Yaskawa INFORM job: X2_24B(90,0).JBI

/JOB
//NAME X2_24B(90,0)
///FOLDERNAME X2
//POS
///NPOS 98,98,98,6,0,0
///TOOL 0
///POSTYPE PULSE
///PULSE
C00000=15575,79859,-14986,13441,104676,73483
C00001=126804,-92055,-48789,28645,51065,65926
C00002=154512,-17095,-20441,46457,51312,77671
C00003=161937,-848,-6352,37251,32753,61979
C00004=159692,17407,12655,41702,31966,59656
C00005=159970,19766,16047,42399,31172,59288
C00006=159972,20330,18267,43630,30372,58648
C00007=159976,20326,18034,43461,30475,58736
C00008=160482,23050,20629,43221,30080,58863
C00009=159976,20326,18034,43461,30475,58736
C00010=159697,17919,14587,42706,31268,59129
C00011=158976,12160,6349,41128,33206,59971
C00012=159418,6486,-154,59703,53174,49617
C00013=160929,10789,6591,60497,51224,48988
C00014=161518,12599,9400,60873,50446,48712
C00015=161521,13127,11564,61641,49913,48166
C00016=161520,13051,11326,61563,49966,48222
C00017=162429,14896,13007,61347,49349,48376
C00018=161520,13051,11326,61563,49966,48222
C00019=160931,11199,8471,61161,50742,48508
C00020=159420,6798,1623,60306,52686,49160
C00021=158595,11215,4105,55963,68819,69684
C00022=160652,12318,8052,56162,66520,69358
C00023=161472,12850,9720,56269,65597,69221
C00024=161473,13383,11888,56662,64989,68781
C00025=161490,13285,11447,56576,65106,68876
C00026=162644,13596,11726,56360,64407,69116
C00027=161490,13285,11447,56576,65106,68876
C00028=160670,12719,9745,56453,66030,69019
C00029=158615,11533,5714,56217,68333,69354
C00030=145844,21981,14022,59749,100145,59975
C00031=147472,19762,14879,59544,98258,59599
C00032=148136,18948,15302,59481,97487,59448
C00033=148138,19507,17514,59327,96919,59020
C00034=148144,19438,17214,59348,96993,59081
C00035=149095,17801,15678,59427,96459,59294
C00036=148144,19438,17214,59348,96993,59081
C00037=147479,20220,16761,59400,97767,59232
C00038=145852,22359,15824,59578,99660,59607
C00039=137889,24717,18086,55155,118108,53390
C00040=138207,19130,15660,54565,117103,52873
C00041=138207,19573,17388,54175,116602,52518
C00042=138207,19438,16874,54289,116751,52623
C00043=138402,17218,14803,54401,116718,52725
C00044=138207,19198,15931,54502,117024,52816
C00045=138380,23714,17318,55251,117790,53487
C00046=145852,22359,15824,59578,99660,59607
C00047=154763,11901,15387,68658,70711,41061
C00048=156717,15177,21386,69242,68625,40420
C00049=157143,15546,21805,69251,68310,40447
C00050=156255,14972,22417,69511,68656,40020
C00051=157248,16273,23616,69515,67962,40120
C00052=157236,16335,23673,69517,67969,40117
C00053=158136,15421,22899,68081,54770,43017
C00054=158597,17339,24094,63812,43421,46704
C00055=158675,18696,25754,61305,36586,48793
C00056=158371,15338,21521,60414,37218,49285
C00057=157215,9529,13249,58606,39045,50279
C00058=155689,128,-5597,51101,67034,60953
C00059=149151,12252,4951,55421,100768,64918
C00060=144904,3935,5079,54220,100687,62374
C00061=145543,-5451,3457,53674,97956,61056
C00062=145117,-2050,7462,53507,97767,60700
C00063=146427,-4037,5767,53710,97024,60980
C00064=153396,2613,11325,54625,92971,62406
C00065=155096,3131,11794,54961,91043,63070
C00066=155127,3166,11823,54964,91024,63076
C00067=158177,1489,10598,55836,83437,65573
C00068=162825,5929,14207,55721,72913,69138
C00069=166488,10840,18435,54134,62935,72728
C00070=165195,8380,15225,53946,63632,72915
C00071=163039,7025,11023,53573,66027,73191
C00072=156115,13997,17270,60701,43178,45173
C00073=157268,19891,25768,62434,41355,44161
C00074=157884,21006,27154,62518,40826,44139
C00075=156967,20197,27277,63317,41176,43618
C00076=158134,20809,27857,62990,40410,43871
C00077=158121,20875,27920,62999,40416,43865
C00078=157099,23447,30366,63399,40803,43589
C00079=155705,26353,33233,56778,30914,48004
C00080=155359,26555,33368,49384,25433,52187
C00081=153014,28261,34997,43179,22329,55472
C00082=153895,25102,30778,39953,22434,57086
C00083=153561,18171,21135,36977,24464,58522
C00084=154328,-437,-7083,34814,53153,69175
C00085=153943,-3670,1993,58187,73110,66585
C00086=156220,-2957,5589,58514,70714,66272
C00087=156644,-2599,7283,58737,69991,66002
C00088=157747,-4828,5565,58281,66085,67202
C00089=157731,-4759,5622,58282,66096,67199
C00090=159511,-232,9113,57226,61670,68810
C00091=163403,5947,13806,51963,49845,73894
C00092=165030,15735,22851,46781,40971,78339
C00093=162686,15609,21777,49814,45504,76092
C00094=160796,11946,15422,49130,47880,76469
C00095=139502,-13197,-17498,52190,59618,73701
C00096=102643,-76138,-42592,31929,63319,59034
C00097=-2000,-92055,-48789,0,51065,0
BC00000=67030,600285,936124
BC00001=198867,566215,454485
BC00002=198867,436418,248072
BC00003=170083,400556,144661
BC00004=170083,415917,144661
BC00005=170083,415917,144661
BC00006=170083,415917,144661
BC00007=170083,415917,144661
BC00008=170083,415917,144661
BC00009=170083,415917,144661
BC00010=170083,415917,144661
BC00011=170083,415917,144661
BC00012=170307,416366,144512
BC00013=170307,416366,144512
BC00014=170307,416366,144512
BC00015=170307,416366,144512
BC00016=170307,416366,144512
BC00017=170307,416366,144512
BC00018=170307,416366,144512
BC00019=170307,416366,144512
BC00020=170307,416366,144512
BC00021=173994,440513,186920
BC00022=173994,440513,186920
BC00023=173994,440513,186920
BC00024=173994,440513,186920
BC00025=173994,440513,186920
BC00026=173994,440513,186920
BC00027=173994,440513,186920
BC00028=173994,440513,186920
BC00029=173994,440513,186920
BC00030=162509,461304,186551
BC00031=162509,461304,186551
BC00032=162509,461304,186551
BC00033=162509,461304,186551
BC00034=162509,461304,186551
BC00035=162509,461304,186551
BC00036=162509,461304,186551
BC00037=162509,461304,186551
BC00038=162509,461304,186551
BC00039=162509,461304,186551
BC00040=162509,461304,186551
BC00041=162509,461304,186551
BC00042=162509,461304,186551
BC00043=162509,461304,186551
BC00044=162509,461304,186551
BC00045=162509,461304,186551
BC00046=162509,461304,186551
BC00047=159532,415917,202070
BC00048=159532,415917,202070
BC00049=159532,415917,202070
BC00050=159532,415917,202070
BC00051=159532,415917,202070
BC00052=159532,415917,202070
BC00053=159532,415917,202070
BC00054=159533,415917,202067
BC00055=159533,415917,202065
BC00056=159532,415917,202070
BC00057=159532,415917,202070
BC00058=177632,434837,235106
BC00059=187185,446552,262931
BC00060=187185,446552,262931
BC00061=187185,446551,262928
BC00062=187185,446551,262928
BC00063=187185,446551,262928
BC00064=187185,446551,262928
BC00065=187185,446552,262930
BC00066=187185,446552,262930
BC00067=187185,446552,262931
BC00068=187185,446552,262931
BC00069=187185,446552,262931
BC00070=187185,446552,262931
BC00071=187185,446552,262931
BC00072=161256,415917,204708
BC00073=161256,415917,204708
BC00074=161256,415917,204708
BC00075=161256,415917,204708
BC00076=161256,415917,204708
BC00077=161256,415917,204708
BC00078=161256,415917,204708
BC00079=161256,415917,204708
BC00080=161256,415917,204708
BC00081=161256,415917,204708
BC00082=161256,415917,204708
BC00083=161256,415917,204708
BC00084=162450,435407,231402
BC00085=163438,443373,249285
BC00086=163438,443373,249285
BC00087=163438,443373,249285
BC00088=163438,443373,249285
BC00089=163438,443373,249285
BC00090=163437,443372,249283
BC00091=163437,443372,249282
BC00092=163437,443372,249282
BC00093=163438,443373,249285
BC00094=163438,443373,249285
BC00095=167011,451779,248072
BC00096=167011,535447,454485
BC00097=198867,523905,632202
EC00000=-798151,-183836
EC00001=-798156,-183832
EC00002=-798156,-183832
EC00003=-798156,-183832
EC00004=-798156,-183832
EC00005=-798156,-183832
EC00006=-798156,-183832
EC00007=-798156,-183832
EC00008=-798156,-183832
EC00009=-798156,-183832
EC00010=-798156,-183832
EC00011=-798156,-183832
EC00012=-798156,-183832
EC00013=-798156,-183832
EC00014=-798156,-183832
EC00015=-798156,-183832
EC00016=-798156,-183832
EC00017=-798156,-183832
EC00018=-798156,-183832
EC00019=-798156,-183832
EC00020=-798156,-183832
EC00021=-798156,-183832
EC00022=-798156,-183832
EC00023=-798156,-183832
EC00024=-798156,-183832
EC00025=-798156,-183832
EC00026=-798156,-183832
EC00027=-798156,-183832
EC00028=-798156,-183832
EC00029=-798156,-183832
EC00030=-798156,-183832
EC00031=-798156,-183832
EC00032=-798156,-183832
EC00033=-798156,-183832
EC00034=-798156,-183832
EC00035=-798156,-183832
EC00036=-798156,-183832
EC00037=-798156,-183832
EC00038=-798156,-183832
EC00039=-798156,-183832
EC00040=-798156,-183832
EC00041=-798156,-183832
EC00042=-798156,-183832
EC00043=-798156,-183832
EC00044=-798156,-183832
EC00045=-798156,-183832
EC00046=-798156,-183832
EC00047=-798156,-183832
EC00048=-798156,-183832
EC00049=-798156,-183832
EC00050=-798156,-183832
EC00051=-798156,-183832
EC00052=-798156,-183832
EC00053=-798156,-183832
EC00054=-798155,-183833
EC00055=-798154,-183833
EC00056=-798156,-183832
EC00057=-798156,-183832
EC00058=-798156,-183832
EC00059=-798156,-183832
EC00060=-798156,-183832
EC00061=-798154,-183833
EC00062=-798154,-183833
EC00063=-798154,-183833
EC00064=-798154,-183833
EC00065=-798155,-183832
EC00066=-798155,-183832
EC00067=-798156,-183832
EC00068=-798156,-183832
EC00069=-798156,-183832
EC00070=-798156,-183832
EC00071=-798156,-183832
EC00072=-798156,-183832
EC00073=-798156,-183832
EC00074=-798156,-183832
EC00075=-798156,-183832
EC00076=-798156,-183832
EC00077=-798156,-183832
EC00078=-798156,-183832
EC00079=-798156,-183832
EC00080=-798156,-183832
EC00081=-798156,-183832
EC00082=-798156,-183832
EC00083=-798156,-183832
EC00084=-798156,-183832
EC00085=-798156,-183832
EC00086=-798156,-183832
EC00087=-798156,-183832
EC00088=-798156,-183832
EC00089=-798156,-183832
EC00090=-798156,-183832
EC00091=-798156,-183832
EC00092=-798156,-183832
EC00093=-798156,-183832
EC00094=-798156,-183832
EC00095=-798156,-183832
EC00096=-798156,-183832
EC00097=-798156,-183832
///POSTYPE BASE
///RECTAN
///RCONF 0,0,0,0,1,0,0,0,0,0,0,0,0,0,0,0,0,0,0,0,0,0,0,0
P00006=2.006,1.622,-0.565,0.0000,0.0000,0.0000
P00021=0.073,2.058,-0.109,0.0000,0.0000,0.0000
P00022=2.006,1.622,-0.565,0.0000,0.0000,0.0000
///RCONF 0,0,0,0,0,0,0,0,0,0,0,0,0,0,0,0,0,0,0,0,0,0,0,0
P00023=-2.957,-4.083,2.762,0.0000,0.0000,0.0000
P00024=-1.466,-0.226,-0.419,0.0000,0.0000,0.0000
P00030=-0.014,-0.768,0.131,0.0000,0.0000,0.0000
//INST
///DATE 2024/12/03 14:06
///ATTR SC,RW
///GROUP1 RB1,BS1
///GROUP2 ST1
NOP
'X2_24B(90,0)
MOVJ C00000 BC00000 VJ=100.00  +MOVJ EC00000 VJ=100.00
MOVJ C00001 BC00001 VJ=100.00  +MOVJ EC00001 VJ=100.00
MOVJ C00002 BC00002 VJ=100.00  +MOVJ EC00002 VJ=100.00
'Path S4187
SSFTOF
SFTOF3D
MOVJ C00003 BC00003 VJ=100.00  +MOVJ EC00003 VJ=100.00
MOVL C00004 BC00004 V=800.0  +MOVJ EC00004 VJ=100.00
SMOVL C00005 BC00005 V=166.7  +MOVJ EC00005
SREFP 3 C00006 BC00006  +REFP EC00006
CALL JOB:SEARCH-R1-S13D
SET P021 P006
SFTON3D P021
SMOVL C00007 BC00007 V=166.7  +MOVJ EC00007
SREFP 3 C00008 BC00008  +REFP EC00008
CALL JOB:SEARCH-R1-S13D
SET P021 P006
SMOVL C00009 BC00009 V=166.7  +MOVJ EC00009
MOVL C00010 BC00010 V=800.0  +MOVJ EC00010 VJ=100.00
MOVL C00011 BC00011 V=1000.0  +MOVJ EC00011 VJ=100.00
'EndPath S4187
'Path S4188
SFTOF3D
MOVJ C00012 BC00012 VJ=100.00  +MOVJ EC00012 VJ=100.00
MOVL C00013 BC00013 V=800.0  +MOVJ EC00013 VJ=100.00
SMOVL C00014 BC00014 V=166.7  +MOVJ EC00014
SREFP 3 C00015 BC00015  +REFP EC00015
CALL JOB:SEARCH-R1-S13D
SET P022 P006
SFTON3D P022
SMOVL C00016 BC00016 V=166.7  +MOVJ EC00016
SREFP 3 C00017 BC00017  +REFP EC00017
CALL JOB:SEARCH-R1-S13D
SET P022 P006
SMOVL C00018 BC00018 V=166.7  +MOVJ EC00018
MOVL C00019 BC00019 V=800.0  +MOVJ EC00019 VJ=100.00
MOVL C00020 BC00020 V=1000.0  +MOVJ EC00020 VJ=100.00
'EndPath S4188
'Path S4189
SFTOF3D
MOVJ C00021 BC00021 VJ=100.00  +MOVJ EC00021 VJ=100.00
MOVL C00022 BC00022 V=800.0  +MOVJ EC00022 VJ=100.00
SMOVL C00023 BC00023 V=166.7  +MOVJ EC00023
SREFP 3 C00024 BC00024  +REFP EC00024
CALL JOB:SEARCH-R1-S13D
SET P023 P006
SFTON3D P023
SMOVL C00025 BC00025 V=166.7  +MOVJ EC00025
SREFP 3 C00026 BC00026  +REFP EC00026
CALL JOB:SEARCH-R1-S13D
SET P023 P006
SMOVL C00027 BC00027 V=166.7  +MOVJ EC00027
MOVL C00028 BC00028 V=800.0  +MOVJ EC00028 VJ=100.00
MOVL C00029 BC00029 V=1000.0  +MOVJ EC00029 VJ=100.00
'EndPath S4189
'Path S4190
SFTOF3D
MOVJ C00030 BC00030 VJ=100.00  +MOVJ EC00030 VJ=100.00
MOVL C00031 BC00031 V=800.0  +MOVJ EC00031 VJ=100.00
SMOVL C00032 BC00032 V=166.7  +MOVJ EC00032
SREFP 3 C00033 BC00033  +REFP EC00033
CALL JOB:SEARCH-R1-S13D
SET P024 P006
SFTON3D P024
SMOVL C00034 BC00034 V=166.7  +MOVJ EC00034
SREFP 3 C00035 BC00035  +REFP EC00035
CALL JOB:SEARCH-R1-S13D
SET P024 P006
SMOVL C00036 BC00036 V=166.7  +MOVJ EC00036
MOVL C00037 BC00037 V=800.0  +MOVJ EC00037 VJ=100.00
MOVL C00038 BC00038 V=1000.0  +MOVJ EC00038 VJ=100.00
'EndPath S4190
'Path W4191
SFTOF3D
SMOVL C00039 BC00039 V=1000.0  +MOVJ EC00039
SMOVL C00040 BC00040 V=166.7  +MOVJ EC00040
SREFP 3 C00041 BC00041  +REFP EC00041
CALL JOB:SEARCH-R1-S13D
SET P030 P006
SFTON3D P030
SMOVL C00042 BC00042 V=166.7  +MOVJ EC00042
SREFP 3 C00043 BC00043  +REFP EC00043
CALL JOB:SEARCH-R1-S13D
SET P030 P006
SMOVL C00044 BC00044 V=250.0  +MOVJ EC00044
SFTOF3D
MOVL C00045 BC00045 V=800.0  +MOVJ EC00045 VJ=100.00
MOVL C00046 BC00046 V=1000.0  +MOVJ EC00046 VJ=100.00
SFTON3D P022
MOVJ C00047 BC00047 VJ=100.00  +MOVJ EC00047 VJ=100.00
SMOVL C00048 BC00048 V=800.0  +MOVJ EC00048
SREFP 1 C00049 BC00049  +REFP EC00049
SREFP 2 C00050 BC00050  +REFP EC00050
SMOVL C00051 BC00051 V=166.7 PL=0  +MOVJ EC00051
MACRO1 MJ#(0) ARGF21
ARCON
SWVON WEV#(100)
SMOVC C00052 BC00052 V=9.2  +MOVJ EC00052
SMOVC C00053 BC00053 V=9.2  +MOVJ EC00053
SMOVC C00054 BC00054 V=9.2  +MOVJ EC00054
SMOVC C00055 BC00055 V=9.2  +MOVJ EC00055
ARCOF
SWVOF
SMOVL C00056 BC00056 V=800.0  +MOVJ EC00056
SMOVL C00057 BC00057 V=1000.0  +MOVJ EC00057
SFTOF3D
'EndPath W4191
MOVJ C00058 BC00058 VJ=100.00  +MOVJ EC00058 VJ=100.00
'Path W4192
SFTOF3D
SSFTOF
SFTON3D P030
MOVJ C00059 BC00059 VJ=100.00  +MOVJ EC00059 VJ=100.00
SMOVL C00060 BC00060 V=800.0  +MOVJ EC00060
SREFP 1 C00061 BC00061  +REFP EC00061
SREFP 2 C00062 BC00062  +REFP EC00062
SMOVL C00063 BC00063 V=166.7 PL=0  +MOVJ EC00063
ARCON
SWVON WEV#(100)
SMOVL C00064 BC00064 V=9.2  +MOVJ EC00064
SMOVL C00065 BC00065 V=9.2  +MOVJ EC00065
SMOVC C00066 BC00066 V=9.2  +MOVJ EC00066
SFTON3D P024
SMOVC C00067 BC00067 V=9.2  +MOVJ EC00067
SMOVC C00068 BC00068 V=9.2  +MOVJ EC00068
SMOVC C00069 BC00069 V=9.2  +MOVJ EC00069
ARCOF
SWVOF
SMOVL C00070 BC00070 V=800.0  +MOVJ EC00070
SMOVL C00071 BC00071 V=1000.0  +MOVJ EC00071
SFTOF3D
'EndPath W4192
'Path W4193
MOVJ C00072 BC00072 VJ=100.00  +MOVJ EC00072 VJ=100.00
SFTON3D P021
SMOVL C00073 BC00073 V=800.0  +MOVJ EC00073
SREFP 1 C00074 BC00074  +REFP EC00074
SREFP 2 C00075 BC00075  +REFP EC00075
SMOVL C00076 BC00076 V=166.7 PL=0  +MOVJ EC00076
ARCON
SWVON WEV#(100)
SMOVC C00077 BC00077 V=9.2  +MOVJ EC00077
SMOVC C00078 BC00078 V=9.2  +MOVJ EC00078
SMOVC C00079 BC00079 V=9.2  +MOVJ EC00079
SMOVC C00080 BC00080 V=9.2  +MOVJ EC00080
SMOVC C00081 BC00081 V=9.2  +MOVJ EC00081
ARCOF
SWVOF
SFTOF3D
SMOVL C00082 BC00082 V=800.0  +MOVJ EC00082
SMOVL C00083 BC00083 V=1000.0  +MOVJ EC00083
'EndPath W4193
MOVJ C00084 BC00084 VJ=100.00  +MOVJ EC00084 VJ=100.00
'Path W4194
MOVJ C00085 BC00085 VJ=100.00  +MOVJ EC00085 VJ=100.00
SMOVL C00086 BC00086 V=800.0  +MOVJ EC00086
SSFTOF
SFTON3D P023
SMOVL C00087 BC00087 V=166.7 PL=0  +MOVJ EC00087
ARCON
SWVON WEV#(100)
SMOVL C00088 BC00088 V=9.2  +MOVJ EC00088
SMOVC C00089 BC00089 V=9.2  +MOVJ EC00089
SMOVC C00090 BC00090 V=9.2  +MOVJ EC00090
SMOVC C00091 BC00091 V=9.2  +MOVJ EC00091
SMOVC C00092 BC00092 V=9.2  +MOVJ EC00092
ARCOF
SWVOF
SFTOF3D
SMOVL C00093 BC00093 V=800.0  +MOVJ EC00093
SMOVL C00094 BC00094 V=1000.0  +MOVJ EC00094
SSFTOF
'EndPath W4194
MOVJ C00095 BC00095 VJ=100.00  +MOVJ EC00095 VJ=100.00
MOVJ C00096 BC00096 VJ=100.00  +MOVJ EC00096 VJ=100.00
MOVJ C00097 BC00097 VJ=100.00  +MOVJ EC00097 VJ=100.00
END
